# EPICS substitutions: ek9000App/Db/EL4112.substitutions
file EL4112.template
{       pattern
        {
                TERMINAL,

        }
        {
        }
}
